// TIA Portal V17 export
// export: Created 2022-07-28T18:03:03.3241752Z, ExportSetting None, DisplayName Totally Integrated Automation Portal, DisplayVersion V17, DisplayName TIA Portal Openness, DisplayVersion V17, DisplayName TIA Portal Teamcenter Gateway, DisplayVersion V17, DisplayName TIA Portal Version Control Interface, DisplayVersion V17, DisplayName TIA Portal Test Suite Advanced, DisplayVersion V17, DisplayName SINAMICS Startdrive Advanced, DisplayVersion V17, DisplayName SINAMICS DCC, DisplayVersion V17, DisplayName SINAMICS Startdrive G130, G150, S120, S150, SINAMICS MV, S210, DisplayVersion V17, DisplayName SINAMICS Startdrive G110M, G120, G120C, G120D, G120P, G115D, DisplayVersion V17, DisplayName STEP 7 Professional, DisplayVersion V17, DisplayName SIMATIC Energy Suite, DisplayVersion V17, DisplayName STEP 7 CFC, DisplayVersion V17, DisplayName STEP 7 Safety, DisplayVersion V17, DisplayName WinCC Advanced / Unified PC, DisplayVersion V17, DisplayName SIMATIC Visualization Architect, DisplayVersion V17
DATA_BLOCK "D_PLC"   // DB1
{ S7_Optimized_Access := 'TRUE' }
// stored: AutoNumber false, InstanceOfName Lib_UDT_PLC, InstanceOfType UDT
"Lib_UDT_PLC"
   // VAR
   //    ID : Int;
   //    CMD : Int;
   //    PLS { S7_SetPoint := 'True'} : "Lib_PLC_PLS";
   //    CycleInfo { S7_SetPoint := 'True'} : "Lib_PLC_CycleInfo";
   //    CMDPRG : UInt;
   //    PRM1 : UInt;
   //    PRM2 : UInt;
   //    Alarm2 : Int;
   //    STEP1 : Int;
   //    T_STEP1 : Int;
   //    Message : UDInt;
   //    NumberDI : Int;
   //    NumberDO : Int;
   //    NumberAI : Int;
   //    NumberAO : Int;
   //    NOW : Array[0..3] of Int;
   //    ShiftParam : Array[0..3] of Int;
   //    ShiftActiveNumber : Int;
   //    TSK_LTIME : LTime;
   //    TSK_MAXTIME : LTime;
   //    TSK_MINTIME : LTime;
   //    TaskTime : "Lib_PLC_TaskTime";
   //    TIME_TCK : Struct
   //       cyclic_sec_R { ExternalVisible := 'False'; ExternalWritable := 'False'} : Real;
   //       cyclic_ms { ExternalVisible := 'False'; ExternalWritable := 'False'} : Int;
   //       cyclic_sec_LR { ExternalVisible := 'False'; ExternalWritable := 'False'} : LReal;
   //       FirstScanTime { ExternalVisible := 'False'; ExternalWritable := 'False'} : Date_And_Time;
   //       PrevScanTime { ExternalVisible := 'False'; ExternalWritable := 'False'} : Date_And_Time;
   //       NowTime { ExternalWritable := 'False'} : Date_And_Time;
   //       Time1cycle_r : LReal;
   //       Time1cycle_di : UDInt;
   //       Time1cycle_DINT : UDInt;
   //       TimeTotalPLC : UDInt;
   //    END_STRUCT;
   //    TaskTime_RUNTIME : Struct
   //       Live : LReal;
   //       TIME_TCK_s : LReal;
   //    END_STRUCT;
   //    MEM_RUNTIME { S7_SetPoint := 'True'} : LReal;
   //    HMI : Struct
   //       State : UDInt;
   //       Alarm : UDInt;
   //       "Counter" : "Lib_PLC_AlarmCounter";
   //    END_STRUCT;
   // END_VAR
BEGIN
END_DATA_BLOCK
